// TwinCAT 3 PLC project POS_Temp_system
// ProgramVersion: 3.1.4022.3
// libraries:
//   CAA Types Extern, * (CAA Technical Workgroup)
//   Tc2_ControllerToolbox, * (Beckhoff Automation GmbH)
//   Tc2_Standard, * (Beckhoff Automation GmbH)
//   Tc2_System, * (Beckhoff Automation GmbH)
//   Tc2_Utilities, * (Beckhoff Automation GmbH)
//   Tc3_Module, * (Beckhoff Automation GmbH)
//   VisuSymbols,3.5.10.0,System
// project tree:
//   DUTs/ SeqState.TcTLEO
//   fbBLOCKS/ fbSensorNoise.TcPOU (not stored), FirstOrder.TcPOU
//   / GlobalTextList.TcGTLO, PlcTask.TcTTO, Visualization Manager.TcVMO (not stored)
//   GVLs/ GVL_IO.TcGVL
//   POUs/ fBDISCRETE_PID.TcPOU, MAIN.TcPOU, POU.TcPOU
//   PROCESSES/ HEATER_PROCESS.TcPOU, SERVO_POS.TcPOU, TANKLEVEL.TcPOU (not stored)
//   VISUs/ UserInterface.TcVIS

CONFIGURATION POS_Temp_system
    RESOURCE PLC ON TwinCAT3
        TASK PlcTask(INTERVAL := T#10ms, PRIORITY := 6);
        PROGRAM MAIN WITH PlcTask : MAIN;
        PROGRAM SERVO_POS WITH PlcTask : SERVO_POS;
        PROGRAM HEATER_PROCESS WITH PlcTask : HEATER_PROCESS;
        PROGRAM TANKLEVEL WITH PlcTask : TANKLEVEL;
    END_RESOURCE
END_CONFIGURATION

// ---- DUTs/SeqState.TcTLEO
{attribute 'qualified_only'}
{attribute 'strict'}
TYPE SeqState :
(
	TO_INIT,
	Ready,
	Fill_A,
	Fill_B,
	Heating,
	ToUnload,
	Drain_1,
	Drain_2
	);
END_TYPE

// ---- GVLs/GVL_IO.TcGVL
{attribute 'qualified_only'}
VAR_GLOBAL
// Process parameters, variables	
	SetPoint_ServoX           :REAL;      // SetPoint X - axis
	SetPointHeater            :REAL;      // SetPoint Heater
	Output_ServoX             :REAL;      // X-axis Position
	Output_Heater             :REAL;      // Temperature Heater
	Output_Stirrer            :BOOL;      // Mixer / Stirrer 
	TankLevelSensor           :REAL;      // Tanklevel analogue sensor 
	ValveA, ValveB, ValveC    :BOOL;      // Valves
	Stirrer					  :BOOL;	  // activate stirrer
	xPushButton1              :BOOL;      // Used for test purposes 
	xPushButton2              :BOOL;      // Used for test purposes
	StartPr, StopPr           :BOOL;      // Start and Stop Process Buttons
	Level_S1,Level_S2,Level_S3:BOOL;      // Level Sensors (digital sensors)
    xGenCtrl_Error            :BOOL;      // General Error due SERVO or HEATER Control          
END_VAR

// ---- POUs/MAIN.TcPOU
PROGRAM MAIN
VAR
	PIDheater_on  : BOOL;  // PID Controller heater enabled ( Closed looop Control)
	PIDServo_on   : BOOL := TRUE;   // PID Controller heater enabled ( Closed looop Control)
	pidServo      : fBDISCRETE_PID;
	pidHeater     : fBDISCRETE_PID;
	States        : SeqState := SeqState.TO_INIT;
	Cmd_Servo     : R_TRIG;
	Cmd_Heater    : R_TRIG;
	Cmd_ProdStart : R_TRIG;
	Cmd_ProdStop  : R_TRIG;
	
	timerA: TP;
	TimA: F_TRIG;
END_VAR

// Handling Buttons
Cmd_ProdStart(clk:=GVL_IO.StartPr);     // Start Process
Cmd_ProdStop(clk:=GVL_IO.StopPr);       // Stop  Process
Cmd_Servo(clk:=GVL_IO.xPushButton1);    // Servo Command button for testing
Cmd_Heater(clk:=GVL_IO.xPushButton2);   // Heater Command button for testing

TimA(clk:=timerA.Q);
timerA();

// ================= START STATE SEQUENCE ======================
//
//   Your State machine program can be programmed here 
//          following an example
//
CASE States OF                       // Sequence State ( ready, etc etc etc )
	//SeqState.Ready:                  // You can change the states if you want for your own convience
	//	GVL_IO.SetPointHeater:= 75;  // Setpoint heater 75 degrees Celsius. 
//	
//SeqState.Fill_A:
		//GVL_IO .ValveA:=TRUE;    //  Open Valve A 	
//	
//

	SeqState.Ready:
	IF GVL_IO.StartPr = TRUE AND GVL_IO.StopPr = FALSE THEN
		GVL_IO.SetPointHeater := 75;
		States := SeqState.Fill_A;
	END_IF
	
	SeqState.TO_INIT:
	GVL_IO.SetPointHeater := 0;
	IF GVL_IO.Output_ServoX > -0.4 AND GVL_IO.Output_ServoX < 0.6 THEN
		PIDServo_on := FALSE;
	ELSE
		GVL_IO.SetPoint_ServoX := 0;
		PIDServo_on := TRUE;
	END_IF
	
	IF GVL_IO.Output_Heater = 0 AND GVL_IO.Level_S1 = TRUE AND GVL_IO.Output_ServoX = 0 THEN
		States := SeqState.Ready;
	END_IF
	
	SeqState.Fill_A:
	GVL_IO.ValveA := TRUE;
	
	IF GVL_IO.Level_S2 = FALSE THEN
		GVL_IO.ValveA := FALSE;
		States := SeqState.Fill_B;
	END_IF
	
	SeqState.Fill_B:
	GVL_IO.ValveB := TRUE;
	PIDheater_on := TRUE;
	GVL_IO.Stirrer := TRUE;
	IF GVL_IO.Level_S3 = FALSE THEN
		GVL_IO.ValveB := FALSE;
		States := SeqState.Heating;
	END_IF
	
	SeqState.Heating:
	IF GVL_IO.Output_Heater > 73.5 AND GVL_IO.Output_Heater < 76.5 THEN
		// turn on timer
		timerA(IN:= TRUE, PT:= T#20S);
		
		// check timer
		IF TimA.Q THEN	
			States := SeqState.ToUnload;
		END_IF
		
	END_IF
	
	SeqState.ToUnload:
	GVL_IO.SetPoint_ServoX := 30;
	PIDServo_on := TRUE;
	
	IF GVL_IO.Output_ServoX > 29.4 AND GVL_IO.Output_ServoX < 30.6 THEN
		PIDServo_on := FALSE;
		PIDheater_on := FALSE;
		States := SeqState.Drain_1;
	END_IF
	
	
	SeqState.Drain_1:
	GVL_IO.ValveC := TRUE;
	IF GVL_IO.Level_S2 = TRUE THEN
		States := SeqState.Drain_2;
	END_IF
	
	SeqState.Drain_2:
	GVL_IO.Stirrer := FALSE;
	IF GVL_IO.Level_S1 = TRUE THEN
		GVL_IO.ValveC := FALSE;
		States := SeqState.TO_INIT;
	END_IF

	
END_CASE
//
//
// ================ END STATE SEQUENCES=========================
// 


// =====   Executing the PID Controllers for  Position and Heater.   ===========
//==================================================================================
//
// *************  Servo with P- Controller only  **************
//
IF (Cmd_Servo.Q AND NOT GVL_IO.xGenCtrl_Error ) THEN
	pidServo.Setpoint:=GVL_IO.SetPoint_ServoX;  // Setpoint Servo
END_IF

pidServo.Kp:= 1;       //  Kp parameter
// pidServo.Ki:= xxx ; //  Ki parameter
// pidServo.Kd:= xxx ; //  Kd parameter 

pidServo.MV_max_sat:= 10;    // Maximum output PID to protect the Servo
pidServo.MV_min_sat:= -10;  // Minimum output PID    ,,     ,,
pidServo.xExt_Error:= Gvl_IO.xGenCtrl_Error;
pidServo.Yprocess:= LREAL_TO_REAL(GVL_IO.Output_ServoX);
//
pidServo(Auto_Mode:=PIDServo_on);  // Calling PID function Heater

// *************   Heater with P- Controller only   **********************
//
IF Cmd_Heater.Q THEN
   pidHeater.Setpoint:=GVL_IO.SetPointHeater;	
END_IF
pidHeater.Kp:= 1;         //  Kp parameter
// pidHeater.Ki:= xx ;    //  Ki parameter     
// pidHeater.Kd:= xx ;    //  Kd parameter      
pidHeater.MV_max_sat:=150;   // Maximum output PID to protect the Heater
pidHeater.MV_min_sat:= -10;  // Minimum output PID ,,     ,,
pidHeater.Yprocess:=GVL_IO.Output_Heater;

pidHeater(Auto_Mode:= PIDheater_on);  // Calling PID function Heater

END_PROGRAM

// ---- POUs/fBDISCRETE_PID.TcPOU
FUNCTION_BLOCK fBDISCRETE_PID
VAR_INPUT
	Setpoint:REAL;         // SetPoint
    Kp:REAL;               // Kp  Proportional gain
	Ki:REAL;               // Ki  Integrated gain
	Kd:REAL;               // Kd  Derivative gain
	Nfilter       : REAL;  // Lowpass Filter Coeff 
	Yprocess      : REAL;  // Process Output
	Auto_Mode     : BOOL;  // PId enable if true (closed loop )
	MV_max_sat    : REAL;  // Maximum Saturation
	MV_min_sat    : REAL;  // Minimum Saturation
	xExt_Error    : BOOL;  // External error 
	
END_VAR
VAR_OUTPUT
	MV_out        : REAL;    // Controller output
	Inposition    : BOOL;    //  2% Settled. not implemented yet. 
END_VAR
VAR
	T1     : REAL :=0;
	Perr, Perr1, Perr2 : REAL ;
    A,B,C  :REAL;
	MV_out1:REAL;
	Tsample:REAL := 0.01;
END_VAR

//
IF T1 = 0 THEN
	MV_out:=0;     // no bias offset controller
END_IF

T1:=Tsample; 
Perr:= Setpoint - Yprocess; // Current error e[k]
//
// Constant Coefficients including the Parameters Kp , Ki, Kd and Tsample
//        Your PID Controller algorithm starts here
//
// A:= (Kp +Ki*(Tsample/2)+(Kd/Tsample));
// B:= (-Kp +Ki*(Tsample/2)-(2*Kd/Tsample));
// C:=  Kd/Tsample;
//
//   Mv_out:= MV_out1 + A*perr +B*perr1 + C*perr2:                                // PID Controller
//
MV_out:=  Kp * Perr;  // P-Controller 

// Update  samples 
MV_out1:= MV_out;      // MV_out[k-1] 
Perr2  := Perr1;       // e[k-2]
Perr1  := Perr;        // e[k-1]

//  PID  is not Enabled 
IF NOT Auto_Mode THEN
	MV_Out:= Setpoint;   ///  Open loop 
END_IF

//    PID  output saturation 
IF Mv_out < MV_min_sat THEN
	Mv_out:= MV_min_sat;
END_IF
IF Mv_out >  MV_max_sat THEN
	Mv_out:= MV_max_sat;
END_IF

END_FUNCTION_BLOCK

// ---- PROCESSES/SERVO_POS.TcPOU
PROGRAM SERVO_POS
VAR CONSTANT
	nTfOrder : USINT := 2;
	nNumOrder : USINT :=2;
	nDenOrder : USINT :=2;
END_VAR
VAR
	aNumArray    : ARRAY[0..nNumOrder] OF FLOAT; //numerator
	aDenArray    : ARRAY[0..nDenOrder] OF FLOAT; //denumerator
	aStructTfData: ARRAY[0..nTfOrder]  OF ST_CTRL_TRANSFERFUNCTION_1_DATA;
	eMode : E_CTRL_MODE;
	stParams : ST_CTRL_TRANSFERFUNCTION_1_PARAMS;
	eErrorId : E_CTRL_ERRORCODES;
	bError : BOOL;
	fbServoX_Tf : FB_CTRL_TRANSFERFUNCTION_1;
	bInit : BOOL := TRUE;
	bPosError:BOOL;
	Tf_Output : LREAL;
	Servo_ERR : R_TRIG;

END_VAR

// IA _Cs4  2019
// O.E Figaroa
// This program simulates a First Order DC Servo with an Integrator
// PLEASE DON'T CHANGE ANY CODE IN THIS PROGRAM !
// Transferfunction Servo Motor X s-domain
//              20
//  Gc =    -----------   [ Theta/u]    and u is proportional to angular position [Theta]
//           0.5s^2 + s 
//
//= = Discrete or z-domain with  Ts = 0.01 s = = 
//          short format
//        0.001987 z + 0.001974
// Gd =  ----------------------   with Ts=0.01 s
//        z^2 - 1.98 z + 0.9802       
// 
//// coefficients obtained by Matlab in long format:
//
// numz =  [0   0.001986733067553   0.001973532271096]     
// denz =  [1.000000000000000 -1.980198673306755   0.980198673306755]
// ==

//========================================
IF bInit THEN
// = numerator ===
aNumArray[0] := 0.001973532271096; 
aNumArray[1] := 0.001986733067553; 
aNumArray[2] := 0.000;
// = denumerator
aDenArray[0] := 0.980198673306755;
aDenArray[1] := -1.980198673306755;
aDenArray[2] := 1.0;
stParams.tTaskCycleTime := T#10MS;
stParams.tCtrlCycleTime := T#10MS;
stParams.nOrderOfTheTransferfunction := nTfOrder;
eMode := eCTRL_MODE_ACTIVE;
bInit := FALSE;
END_IF
stParams.pNumeratorArray_ADR := ADR(aNumArray);
stParams.nNumeratorArray_SIZEOF := SIZEOF(aNumArray);
stParams.pDenominatorArray_ADR := ADR(aDenArray);
stParams.nDenominatorArray_SIZEOF := SIZEOF(aDenArray);
stParams.pTransferfunction1Data_ADR := ADR(aStructTfData);
stParams.nTransferfunction1Data_SIZEOF := SIZEOF(aStructTfData);

// Execute TF 

fbServoX_Tf (fIn :=main.pidServo.MV_out,
eMode := eMode,
stParams := stParams,
fOut => Tf_Output,
eErrorId => eErrorId,
bError => bError);

GVL_IO.Output_ServoX:=LREAL_TO_REAL(fbServoX_Tf.fOut);	

Servo_ERR(CLK:=(ABS(GVL_IO.Output_ServoX) > 50),Q=>GVL_IO.xGenCtrl_Error);

END_PROGRAM

// ---- PROCESSES/HEATER_PROCESS.TcPOU
PROGRAM HEATER_PROCESS
VAR CONSTANT
	nTfOrder : USINT := 2;
	nNumOrder : USINT :=2;
	nDenOrder : USINT :=2;
END_VAR
VAR
	aNumArray        : ARRAY[0..nNumOrder] OF FLOAT; //numerator
	aDenArray        : ARRAY[0..nDenOrder] OF FLOAT; //denumerator
	aStructTfData    : ARRAY[0..nTfOrder]  OF ST_CTRL_TRANSFERFUNCTION_1_DATA;
	eMode            : E_CTRL_MODE;
	stParams         : ST_CTRL_TRANSFERFUNCTION_1_PARAMS;
	eErrorId         : E_CTRL_ERRORCODES;
	bError           : BOOL;
	fbHeater_Tf      : FB_CTRL_TRANSFERFUNCTION_1;
	bInit            : BOOL := TRUE;
	Tfunction_Input  : FLOAT := 0;
	Setpoint_Heater  : INT;
	Tf_Heater_Output : LREAL;
   
END_VAR

// IA _Cs4  2019
// O.E Figaroa
// This program simulates a Second Order Process aka Heater Process.
// PLEASE DON'T CHANGE ANY CODE IN THIS PROGRAM !
// Transferfunction Heater
//                  5
///  G(s)=  ---------------------    [ Temp / Temp ]
//          256 s^2 + 100 s + 5
//= = = = = = = = = = = = = = = = 
// Discrete transfer function of the Heater
//
//
//          9.753E-07 z + 9.74E-07
// G(z)=  ----------------------
//          z^2 - 1.996 z + 0.9961
//
// Obtained coefficients in long formats for accuracy purposes
//
// numerator =    1.0e-06 * [0   0.975292016341129   0.974022931328863]
// denumerator = [1.000000000000000  -1.996099420155170   0.996101369470118]

IF bInit THEN
// = numerator ===
aNumArray[0] := 0.974022931328863 * 1E-06;
aNumArray[1] := 0.975292016341129 * 1E-06;
aNumArray[2] := 0.000;
// = denumerator
aDenArray[0] := 0.996101369470118;
aDenArray[1] := -1.996099420155170;
aDenArray[2] := 1.00000;
// 

stParams.tTaskCycleTime := T#10MS;
stParams.tCtrlCycleTime := T#10MS;
stParams.nOrderOfTheTransferfunction := nTfOrder;
eMode := eCTRL_MODE_ACTIVE;
bInit := FALSE;
END_IF

stParams.pNumeratorArray_ADR := ADR(aNumArray);
stParams.nNumeratorArray_SIZEOF := SIZEOF(aNumArray);
stParams.pDenominatorArray_ADR := ADR(aDenArray);
stParams.nDenominatorArray_SIZEOF := SIZEOF(aDenArray);
stParams.pTransferfunction1Data_ADR := ADR(aStructTfData);
stParams.nTransferfunction1Data_SIZEOF := SIZEOF(aStructTfData);
// Execute TF 
fbHeater_Tf (fIn := main.pidHeater.MV_out,
eMode := eMode,
stParams := stParams,
fOut => Tf_Heater_Output,
eErrorId => eErrorId,
bError => bError);
//
GVL_IO.Output_Heater:=LREAL_TO_REAL(fbHeater_Tf.fOut );
IF fbHeater_Tf.fOut <= 0 THEN
	GVL_IO.Output_Heater:=0;
END_IF

END_PROGRAM

// ---- fbBLOCKS/FirstOrder.TcPOU
FUNCTION_BLOCK FirstOrder
VAR_INPUT
	Gain: REAL;
	Tconstant : REAL;
	fBIn   : REAL;
END_VAR
VAR_OUTPUT
	fBOut  : REAL;
END_VAR
VAR
	ssy, Sy   :REAL;
	Tsample: REAL := 0.01;
END_VAR

// This program simulates a First Order Euler Emulation
// PLEASE DON'T CHANGE ANY CODE IN THIS PROGRAM !
// Euler Emulation 1st Order with 0.01 sec sampletime.
sy := ( fBIn * Gain / Tconstant ) - ( fBOut / Tconstant ) ;
fBOut := fBout + ( sy * Tsample ) ;

END_FUNCTION_BLOCK

// ---- POUs/POU.TcPOU
FUNCTION_BLOCK POU
VAR_INPUT
END_VAR
VAR_OUTPUT
END_VAR
VAR
END_VAR

// NETWORK 1

END_FUNCTION_BLOCK

// ---- GlobalTextList.TcGTLO
TEXTLIST GlobalTextList
  249 = '%.1d'
  0 = '%.1f'
  112 = '%.2f'
  438 = '%d'
  47 = 'Auto-Mode Heater'
  280 = 'Auto-Mode Servo'
  694 = 'Auto-Modee Servo'
  753 = 'Drain Position'
  601 = 'Home'
  167 = 'Outlet'
  445 = 'Output Heater   %.2f'
  735 = 'Output PID  %.2f'
  160 = 'Output Servo   %.2f'
  940 = 'Overshoot'
  350 = 'Overshoot= 30'
  17 = 'PID-Enable'
  786 = 'PID-Enable Heater'
  168 = 'PID-Enable Servo'
  520 = 'Position %s'
  468 = 'Position = 0'
  917 = 'Position = 30'
  409 = 'Position and Temperature Control in Batch Process'
  224 = 'Position and Temperature Control in Batch Processes'
  93 = 'Response %s'
  81 = 'Response X -axis %s'
  617 = 'Response X -axis:   %s'
  12 = 'Response Y -axis %s'
  134 = 'Response Y -axis:   %s'
  150 = 'Servo Error'
  621 = 'Servo Running CCW'
  147 = 'Setpoint %.2f'
  636 = 'SetPoint %s'
  401 = 'Setpoint Heater   %.2f'
  352 = 'Setpoint Servo   %.2f'
  368 = 'SetPoint: %d'
  75 = 'SetPoint: %s'
  637 = 'SP Heater cmd'
  808 = 'SP Servo cmd'
  389 = 'START'
  433 = 'STOP'
  527 = 'Tank'
  652 = 'TANK'
  181 = 'Tanklevel Sensor:    %.2f'
  276 = 'Tanklevel:    %.2f'
  119 = 'Unload  Position'
  434 = 'Wall HIT !'
END_TEXTLIST

// ---- VISUs/UserInterface.TcVIS
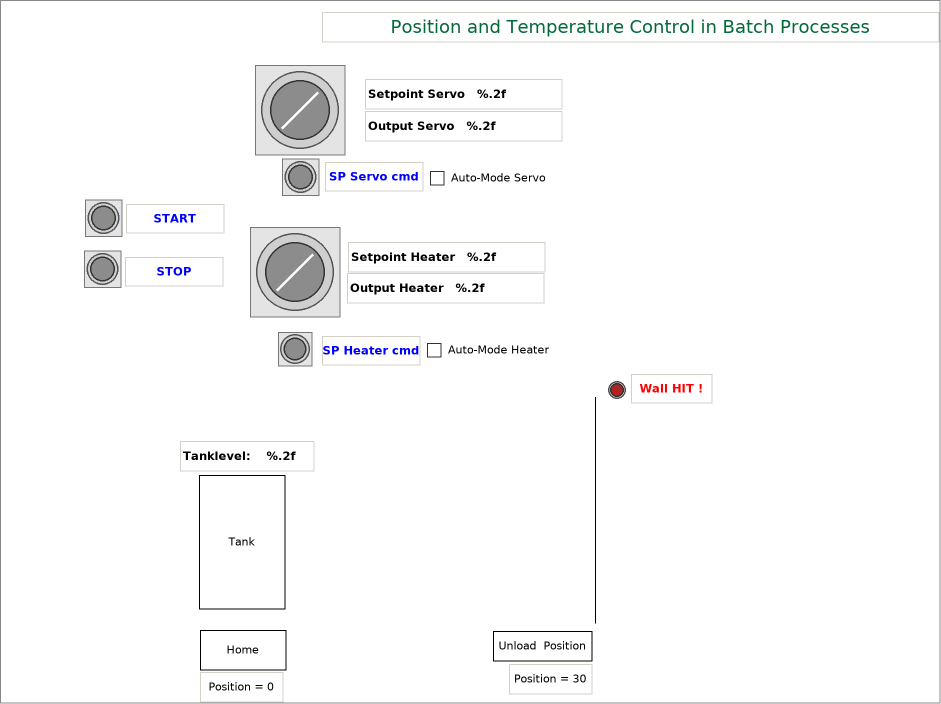
VISUALIZATION UserInterface  // 941x704
    PushSwitch (282,158 37x38), variable: GVL_IO.xPushButton1, behaviour: TAP, style: Switch-PushSwitch-Gray
    Potentiometer360 (255,65 90x90), variable: GVL_IO.SetPoint_ServoX, style: Potentiometer-Potentiometer360-Gray, scale format: %d, scale 0..60
        p2431819421: Outside
    Textfield (365,79 197x30), "Setpoint Servo %.2f", text variable: GVL_IO.SetPoint_ServoX
    Textfield (365,111 197x30), "Output Servo %.2f", text variable: GVL_IO.Output_ServoX
    Potentiometer360 (250,227 90x90), variable: GVL_IO.SetPointHeater, style: Potentiometer-Potentiometer360-Gray, scale format: %d, scale 0..100
        p2431819421: Outside
    PushSwitch (278,331 34x36), variable: GVL_IO.xPushButton2, behaviour: TAP, style: Switch-PushSwitch-Gray
    Textfield (348,242 197x30), "Setpoint Heater %.2f", text variable: GVL_IO.SetPointHeater
    Textfield (347,273 197x30), "Output Heater %.2f", text variable: GVL_IO.Output_Heater
    Rectangle (200,630 86x40), "Home"
    Rectangle (493,631 99x30), "Unload Position"
    Textfield (509,664 83x30), "Position = 30"
    Textfield (200,672 83x30), "Position = 0"
    Rectangle (199,475 86x134), "Tank"
        p3560616238: GVL_IO.Output_ServoX * 10
    Textfield (322,336 98x29), "SP Heater cmd"
    Textfield (325,162 98x29), "SP Servo cmd"
    Textfield (322,12 617x30), "Position and Temperature Control in Batch Processes"
    Textfield (180,441 134x30), "Tanklevel: %.2f", text variable: GVL_IO.TankLevelSensor
    Checkbox (425,340 125x20), "Auto-Mode Heater", variable: MAIN.PIDheater_on
    Checkbox (428,168 129x20), "Auto-Mode Servo", variable: MAIN.PIDServo_on
    Line (595,397) (595,623)
    Lamp1 (607,380 20x20), variable: (GVL_IO.Output_ServoX>31), style: Lamp-Lamp1-Red
    Textfield (631,374 81x29), "Wall HIT !", invisible if: (GVL_IO.Output_ServoX<=30.6)
    PushSwitch (85,199 37x38), variable: GVL_IO.StartPr, behaviour: TAP, style: Switch-PushSwitch-Gray
    PushSwitch (84,250 37x38), variable: GVL_IO.StopPr, behaviour: TAP, style: Switch-PushSwitch-Gray
    Textfield (126,204 98x29), "START"
    Textfield (125,257 98x29), "STOP"
END_VISUALIZATION
